FUNCTION_BLOCK FB_ST10
VAR
	_camera : BOOL;
	_triger : BOOL;
	_description : STRING;
	_test : BOOL;
	_cameraProgram : UINT;
	_gitTest : BOOL;
	_git : INT;
	_ivana : INT;
END_VAR

METHOD PROTECTED _camera
VAR_INPUT
END_VAR
IF _camera THEN 
	_description:= 'On';
ELSE 
	_triger:= TRUE; 
END_IF
END_METHOD

METHOD _scanner : BOOL
VAR_INPUT
END_VAR
IF _triger THEN 
	_description:= 'Trger scanner';
END_IF
_gitTest:= TRUE; 
_ivana := 5;
END_METHOD

END_FUNCTION_BLOCK

(* stored: Version 1.1.0.1, ProductVersion 3.1.4024.12
   POU FB_ST10: Id {61144e30-0e02-44e4-a1c9-c2000a6e1c68}, SpecialFunc None
   Method _camera: Id {607f1da7-acd9-442b-8e19-2806946f35ab}
   Method _scanner: Id {4ecb456b-c5dd-44ea-a517-3dca9868e0e9} *)
